DATA_BLOCK "DB_Plc_RouteFsmWork"
{ S7_Optimized_Access := 'TRUE' }
VERSION : 0.1

VAR
  RoutesWork : ARRAY[1..12] OF "UDT_RouteFsmWork";
END_VAR

BEGIN
END_DATA_BLOCK
